// TIA Portal V19 export
FUNCTION "AnalogReadValues" : Void   // FC8, STL
TITLE = Read Analog Input Value
{ S7_Optimized_Access := 'TRUE' }
VERSION : 0.0
// Comment
// stored: AutoNumber false
BEGIN

NETWORK
TITLE = Read Analog Input Value, TT01.76
// CALL  "ANA.ANALOG READING (SYS)"
//        IN_INT  :="TT0176"
//        MAX_REAL:=1.600000e+003
//        MIN_REAL:=0.000000e+000
//        OUT_REAL:="DB-ANALOG INPUT".TT0176REAL
//        OUT_INT :="DB-ANALOG INPUT".TT0176MEAS
      CALL  "AnalogReadingSystem"
      ( IN_PIW   := "P_TT0176":P,
        MAX_REAL := 160.0,
        MIN_REAL := 0.0,
        OUT_REAL := "MeasuredValues".TT0176REAL
      );


NETWORK
TITLE = Read Analog Input Value, TT01.78
// CALL  "ANA.ANALOG READING (SYS)"
//        IN_INT  :="TT0178"
//        MAX_REAL:=1.600000e+003
//        MIN_REAL:=0.000000e+000
//        OUT_REAL:="DB-ANALOG INPUT".TT0178REAL
//        OUT_INT :="DB-ANALOG INPUT".TT0178MEAS
      CALL  "AnalogReadingSystem"
      ( IN_PIW   := "P_TT0178":P,
        MAX_REAL := 160.0,
        MIN_REAL := 0.0,
        OUT_REAL := "MeasuredValues".TT0178REAL
      );


NETWORK
TITLE = Read Analog Input Value, TT01.60
// CALL  "ANA.ANALOG READING (SYS)"
//        IN_INT  :="TT0160"
//        MAX_REAL:=1.600000e+003
//        MIN_REAL:=0.000000e+000
//        OUT_REAL:="DB-ANALOG INPUT".TT0160REAL
//        OUT_INT :="DB-ANALOG INPUT".TT0160MEAS
      CALL  "AnalogReadingSystem"
      ( IN_PIW   := "P_TT0160":P,
        MAX_REAL := 160.0,
        MIN_REAL := 0.0,
        OUT_REAL := "MeasuredValues".TT0160REAL
      );


NETWORK
TITLE = Read Analog Input Value, TT01.72
// CALL  "ANA.ANALOG READING (SYS)"
//        IN_INT  :="TT0172"
//        MAX_REAL:=1.600000e+003
//        MIN_REAL:=0.000000e+000
//        OUT_REAL:="DB-ANALOG INPUT".TT0172REAL
//        OUT_INT :="DB-ANALOG INPUT".TT0172MEAS
      CALL  "AnalogReadingSystem"
      ( IN_PIW   := "P_TT0172":P,
        MAX_REAL := 160.0,
        MIN_REAL := 0.0,
        OUT_REAL := "MeasuredValues".TT0172REAL
      );


NETWORK
TITLE = Read Analog Input Value, TT01.63
// LOAD 1300 (130.0 CELSIUS) IF NO AGITATOR IS CONNECTED
//     CALL  "ANA.ANALOG READING (SYS)"
//        IN_INT  :="TT0180"
//        MAX_REAL:=1.600000e+003
//        MIN_REAL:=0.000000e+000
//        OUT_REAL:="DB-ANALOG INPUT".TT0163REAL
//        OUT_INT :="DB-ANALOG INPUT".TT0163MEAS
      L     130.0;  // no TT 01.63 present
      T     "MeasuredValues".TT0163REAL;


NETWORK
TITLE = Read Analog Input Value, TT01.80
// CALL  "ANA.ANALOG READING (SYS)"
//        IN_INT  :="TT0180"
//        MAX_REAL:=1.600000e+003
//        MIN_REAL:=0.000000e+000
//        OUT_REAL:="DB-ANALOG INPUT".TT0180REAL
//        OUT_INT :="DB-ANALOG INPUT".TT0180MEAS
      CALL  "AnalogReadingSystem"
      ( IN_PIW   := "P_TT0180":P,
        MAX_REAL := 160.0,
        MIN_REAL := 0.0,
        OUT_REAL := "MeasuredValues".TT0180REAL
      );


NETWORK
TITLE = Read Analog Input Value, PT01.67
// REMEMBER TO DIVIDE REAL VALUE WITH 100 
//       CALL  "ANA.ANALOG READING (SYS)"
//        IN_INT  :="PT0167"
//        MAX_REAL:=6.000000e+002
//        MIN_REAL:=0.000000e+000
//        OUT_REAL:="DB-ANALOG INPUT".PT0167REAL
//        OUT_INT :="DB-ANALOG INPUT".PT0167MeasPressure
// //
//       L     "DB-ANALOG INPUT".PT0167REAL
//       L     1.000000e+002
//       /R    
//       T     "DB-ANALOG INPUT".PT0167REAL
      CALL  "AnalogReadingSystem"
      ( IN_PIW   := "P_PT0167":P,
        MAX_REAL := 6.0,
        MIN_REAL := 0.0,
        OUT_REAL := "MeasuredValues".PT0167REAL
      );


NETWORK
TITLE = Read Analog Input Value, WT01.69
// REMEBER TO ENTER ACTUAL SIZE OF A-TANK
// EXAMPLE: WEIGHING CELL 0-10.000 KG, THREE LEGS
//          MAX_REAL:= 30.000 KG   
// //
//       CALL  "ANA.ANALOG READING (SYS)"
//        IN_INT  :="WT0169"
//        MAX_REAL:=1.500000e+004          // WEIGHING CELL 0-10 TON ~ SCALING 
// 30000 KG
//        MIN_REAL:=0.000000e+000
//        OUT_REAL:="DB-ANALOG INPUT".WT0169REAL
//        OUT_INT :="DB-ANALOG INPUT".WT0169MeasWeight
      CALL  "AnalogReadingSystem"
      ( IN_PIW   := "P_WT0169":P,
        MAX_REAL := 15000.0,
        MIN_REAL := 0.0,
        OUT_REAL := "MeasuredValues".WT0169REAL
      );

//    L     2.900000e+002               //zero correction
//    L     "MeasuredValues".WT0169REAL
//     +R
//      T     "MeasuredValues".WT0169REAL



NETWORK
TITLE = Read Analog Input Value, CT01.82
// CT01.82 CIP RETURN CONTRATION 
// //
//       CALL  "ANA.ANALOG READING (SYS)"
//        IN_INT  :="CT0182"
//        MAX_REAL:=2.500000e+002
//        MIN_REAL:=0.000000e+000
//        OUT_REAL:="DB-ANALOG INPUT".CT0182REAL
//        OUT_INT :="DB-ANALOG INPUT".CT0182MEAS
      CALL  "AnalogReadingSystem"
      ( IN_PIW   := "P_CT0182":P,
        MAX_REAL := 250.0,
        MIN_REAL := 0.0,
        OUT_REAL := "MeasuredValues".CT0182REAL
      );

NETWORK
TITLE = 
      CALL  "AnalogReadingSystem"
      ( IN_PIW   := "P_TT0950":P,
        MAX_REAL := 200.0,
        MIN_REAL := 0.0,
        OUT_REAL := "MeasuredValues".TT0950REAL
      );


NETWORK
TITLE = 
      CALL  "AnalogReadingSystem"
      ( IN_PIW   := "P_TT0951":P,
        MAX_REAL := 200.0,
        MIN_REAL := 0.0,
        OUT_REAL := "MeasuredValues".TT0951REAL
      );

END_FUNCTION
